{attribute 'qualified_only'}
VAR_GLOBAL
	// Create this Folder to store log
	Log_Directory : STRING := 'C:\Users\celli\OneDrive\Desktop\TEST_LOG\PROCESS\';
END_VAR

VAR_GLOBAL PERSISTENT
	yesterday 	: STRING;
	today		: STRING;
END_VAR

(* stored: Version 1.1.0.1, ProductVersion 3.1.4024.12
   GVL GVL: Id {3536f781-1aba-490f-bf6b-e5c225871912} *)
